FUNCTION_BLOCK Reset1
VAR_INPUT
	Execute : BOOL;
END_VAR
VAR_OUTPUT
	Done : BOOL;
END_VAR
VAR
	PickParams: PickPars_typ;
	gState: INT;
	iMovementNumber: INT;
END_VAR

Done := FALSE;
(*
IF Execute THEN
	CASE gState OF
	300: // Dump Puck
			iMovementNumber := 8;
			Delta.MoveDirectTo( GVL.DeltaCoords[iMovementNumber].x, GVL.DeltaCoords[iMovementNumber].y, GVL.DeltaCoords[iMovementNumber].z);		
			gState := 330;
			iMovementNumber := 9;
		
	330:
			IF Delta.MovePathDone THEN
			Delta.MoveDirectTo( GVL.DeltaCoords[iMovementNumber].x, GVL.DeltaCoords[iMovementNumber].y, GVL.DeltaCoords[iMovementNumber].z);			
				gState := 332;	
			END_IF
	332:
	
			IF Delta.MovePathDone THEN
				Delta.DisableAir();
				gState := 335;
			END_IF
			
	335:
			Delta.MoveDirectTo( GVL.DeltaCoords[iMovementNumber].x, GVL.DeltaCoords[iMovementNumber].y, GVL.DeltaCoords[iMovementNumber].z + 25);			
			gState := 340;
	340:
			IF Delta.MovePathDone THEN
			//	SystemCommands.MoverRelease := TRUE;
				Done := TRUE;		
			END_IF	
	END_CASE
ELSE
	gState := 300;
	Done := FALSE;
END_IF	*)

END_FUNCTION_BLOCK

(* stored: Version 1.1.0.1, ProductVersion 3.1.4024.11
   POU Reset1: Id {2268c0fe-288a-4490-aa7d-0ba072bf20b2}, SpecialFunc None *)
